{attribute addProperty BoxType "AT2041-0250-0021"}
{attribute addProperty Id "A_0101_AT2041_5250_0018_AT2041_5250AT2041_C5E5984862678.25"}
{attribute addProperty CRC "957722665"}
{attribute addProperty SizeInBites "626"}
{attribute addProperty SizeInBytes "78.25"}
TYPE A_0043_AT2041_0250_0021_3915B029 EXTENDS AT2041_BA5A9548 :
STRUCT
	{attribute addProperty Name "A_0101_AT2041_5250_0018_AT2041_5250"}
	A_0101_AT2041_5250_0018_AT2041_5250 : AT2041_C5E59848;
END_STRUCT
END_TYPE

(* stored: Version 1.2.0.0, ProductVersion 3.1.4024.9
   DUT A_0043_AT2041_0250_0021_3915B029: Id {985cc429-8702-4798-923f-3c14148e3357} *)
